TYPE StrPathName_t : String(255); END_TYPE

(* stored: Version 1.1.0.1, ProductVersion 3.1.4024.12
   DUT StrPathName_t: Id {f7906ba5-63c0-45a1-8fcb-e419b849bbdb} *)
